Omron CX-Programmer project NewProject (CX-Programmer 9.81)

# PLC Latch: CJ1M CPU11

## Program NewProgram1 (cyclic task 0)
Local symbols
BE 0.00 BOOL  ; Botao emer
BS 0.01 BOOL  ; botao stop
Bstart 0.02 BOOL  ; botao start
KM1 0.03 BOOL  ; KM1
KM2 0.06 BOOL  ; km2
KM_1 0.03 BOOL  ; out
NO2_KM1 0.03 BOOL  ; NO2KM1
NO_KM2 0.06 BOOL  ; noKM2

### Section Section1

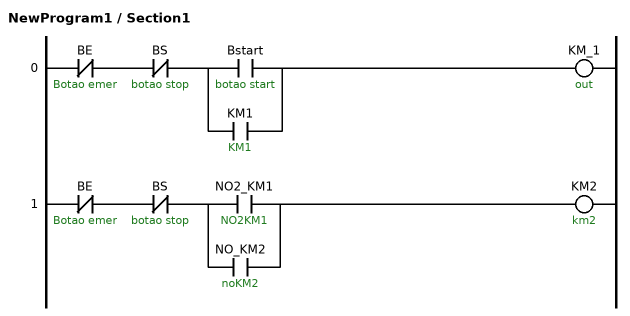
; rung 0
LDNOT BE  ; Botao emer
ANDNOT BS  ; botao stop
LD Bstart  ; botao start
OR KM1  ; KM1
ANDLD
OUT KM_1  ; out
; rung 1
LDNOT BE  ; Botao emer
ANDNOT BS  ; botao stop
LD NO2_KM1  ; NO2KM1
OR NO_KM2  ; noKM2
ANDLD
OUT KM2  ; km2

### Section END
; rung 0
END(001)